(* CODESYS project Prova_CTU.project

Project tree, tasks and I/O mapping:
  Device : CODESYS Control Win V3, 3S - Smart Software Solutions GmbH, order no. 305021, version 3.5.10.30
    application Application
      libraries: Standard, * (System)
      task MainTask (cyclic, interval t#20ms, priority 1) calls PLC_PRG
      task VISU_TASK (cyclic, interval 100 ms, priority 31) calls VisuElems.Visu_Prg
      program PLC_PRG [FBD]
      visualisation Visualization
  text list GlobalTextList
*)

// Device/Application/PLC_PRG
PROGRAM PLC_PRG
VAR
	Contact1: BOOL := FALSE;
	Coil1: BOOL := FALSE;
	PV1: WORD := 3;
	CTU_0: CTU;
	CV: WORD;
END_VAR

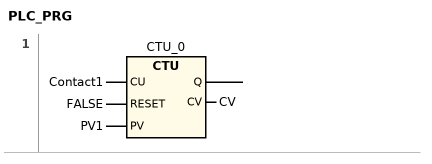
// NETWORK 1
CTU_0(CU := Contact1, RESET := FALSE, PV := PV1, CV => CV); // CTU

END_PROGRAM

// Device/Application/Visualization
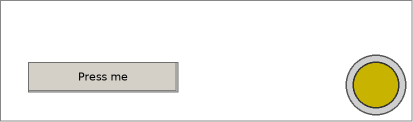
VISUALIZATION Visualization  // 413x122
    Lamp1 (341,50 70x70), variable: PLC_PRG.CTU_0.Q, style: Lamp-Lamp1-Yellow
    Button (28,62 150x30), "Press me"
        tap PLC_PRG.Contact1
END_VISUALIZATION
